{attribute 'qualified_only'}
{attribute 'strict'}
TYPE eSubValues :
(
	Minimum := 0,
	Average := 1,
	Maximum := 2
);
END_TYPE

(* stored: Version 1.1.0.1, ProductVersion 3.1.4024.12
   DUT eSubValues: Id {c90aa7e7-15ee-4088-952d-0f4bbf685883} *)
